TYPE ST_System_Fenster_Parameter :
STRUCT
	Zeit_Stellen1			: DINT;
	Zeit_Stellen0			: DINT;

	AutoQuittierung			: BOOL;
END_STRUCT
END_TYPE

(* stored: Version 1.1.0.1, ProductVersion 3.1.4024.9
   DUT ST_System_Fenster_Parameter: Id {e23950e7-6f8a-4a39-a1ed-0f31d5af880c} *)
